(* Logix 5000 project; controller LeakTestAuto vendor 1 type 14 code 226 rev 37.11; software revision 37.01; part 14 of 15 *)
(* tags used below, declared in another part *)
   AOI_CapActuators_Seq : AOI_Sequencer_x64;
   AOI_CapCTS_Seq : AOI_Sequencer_x64;
   AOI_CapFail_Seq : AOI_Sequencer_x64;
   AOI_CapRobot_Seq : AOI_Sequencer_x64;
   AOI_CTS1 : AOI_CTS_INSTRUMENT;
   AOI_CTS2 : AOI_CTS_INSTRUMENT;
   AOI_RobotPos : AOI_RobotPositions;
   AOI_SeqSteps : AOI_StandardSeqSteps;
   AOI_SRX100 : AOI_KeyenceBarcode;
   BarcodeScanner : udt_OutputStructure;
   CapActuators_BarcodeBad : COUNTER;
   CapActuators_BarcodeGood : COUNTER;
   CapActuators_CTS1Bad : COUNTER;
   CapActuators_CTS1Good : COUNTER;
   CapActuators_CTS2Bad : COUNTER;
   CapActuators_CTS2Good : COUNTER;
   CapActuators_Nest1HasPart : BOOL;
   CapActuators_Nest2HasPart : BOOL;
   CapActuators_Seq : udt_SequenceStructure_X64;
   CapCTS_CTS1Bad : COUNTER;
   CapCTS_CTS1Good : COUNTER;
   CapCTS_CTS2Bad : COUNTER;
   CapCTS_CTS2Good : COUNTER;
   CapCTS_Nest1HasPart : BOOL;
   CapCTS_Nest2HasPart : BOOL;
   CapCTS_Seq : udt_SequenceStructure_X64;
   CapFail_Seq : udt_SequenceStructure_X64;
   CapRobot_IsNest : BOOL;
   CapRobot_Seq : udt_SequenceStructure_X64;
   CapRobot_StartPos : DINT;
   CapRobot_TargetPos : DINT;
   CapShuffle_Seq : udt_SequenceStructure_X64;
   Conveyor : udt_OutputStructure;
   Conveyor_Seq : udt_SequenceStructure_X64;
   LeakTester1 : udt_OutputStructure;
   LeakTester2 : udt_OutputStructure;
   Nest1Cylinder : udt_OutputStructure;
   Nest2Cylinder : udt_OutputStructure;
   OP220 : udt_Mode;
   Robot : udt_OutputStructure;
   RobotGripper : udt_OutputStructure;
   RobotInputs : udt_EpsonInputs;
   TempConsumedFromPLC : BOOL;
   TON_CapActuatorsDelay : TIMER;
   TON_CapActuatorsDelay2 : TIMER;
   TON_CapCTSDelay : TIMER;
   TON_CapCTSDelay2 : TIMER;
   TON_FailChute : TIMER[10];
   I_OP220_N3_CONVEYOR_LOAD : ALIAS FOR Local:3:I.Pt12.Data;
   I_OP220_N3_DUT_PRE_NEST_0 : ALIAS FOR Local:3:I.Pt00.Data;
   I_OP220_N3_DUT_PRE_NEST_1 : ALIAS FOR Local:3:I.Pt01.Data;
   I_OP220_N3_DUT_PRE_NEST_2 : ALIAS FOR Local:3:I.Pt02.Data;
   I_OP220_N3_NEST1_EXTEND : ALIAS FOR Local:3:I.Pt04.Data;
   I_OP220_N3_NEST1_HOME : ALIAS FOR Local:3:I.Pt03.Data;
   I_OP220_N3_NEST2_EXTEND : ALIAS FOR Local:3:I.Pt06.Data;
   I_OP220_N3_NEST2_HOME : ALIAS FOR Local:3:I.Pt05.Data;
   I_OP220_N3_REJECT_CHUTE_PART : ALIAS FOR Local:3:I.Pt10.Data;
   PLC : AOI_PLC;
(* MainProgram, continued *)

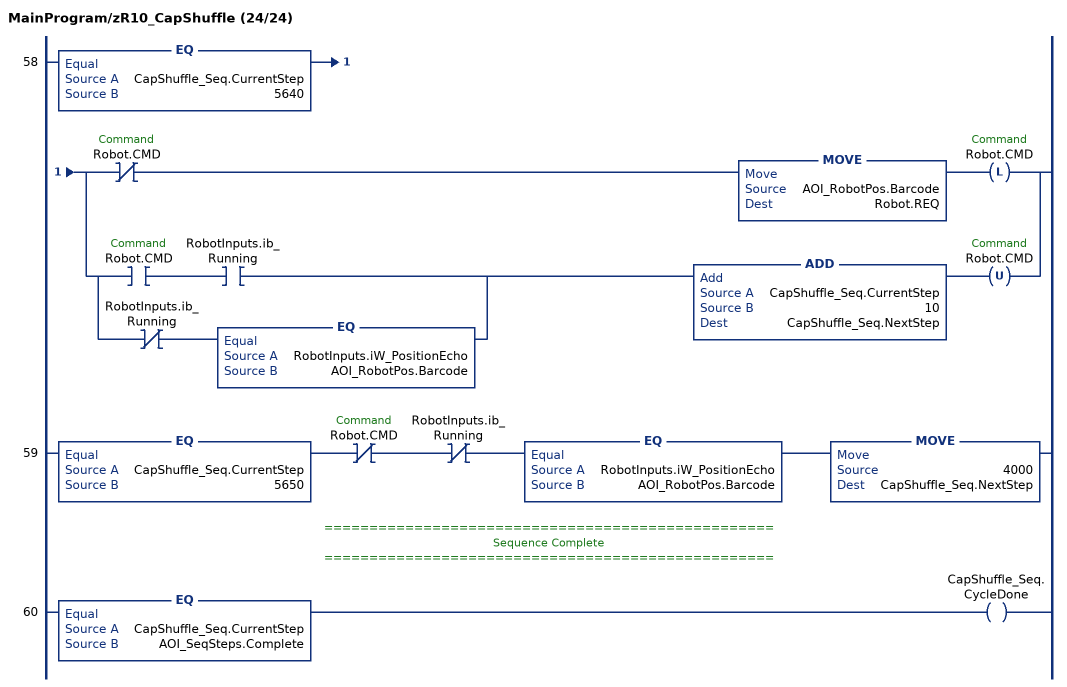
   [picture p173: MainProgram/zR10_CapShuffle rungs 58-60]
   58: EQ(CapShuffle_Seq.CurrentStep,5640)[XIO(Robot.CMD) MOVE(AOI_RobotPos.Barcode,Robot.REQ) OTL(Robot.CMD) ,[XIC(Robot.CMD) XIC(RobotInputs.ib_Running) ,XIO(RobotInputs.ib_Running) EQ(RobotInputs.iW_PositionEcho,AOI_RobotPos.Barcode) ] ADD(CapShuffle_Seq.CurrentStep,10,CapShuffle_Seq.NextStep) OTU(Robot.CMD) ];
   59: EQ(CapShuffle_Seq.CurrentStep,5650)XIO(Robot.CMD)XIO(RobotInputs.ib_Running)EQ(RobotInputs.iW_PositionEcho,AOI_RobotPos.Barcode)MOVE(4000,CapShuffle_Seq.NextStep);
   // ==================================================
   // Sequence Complete
   // ==================================================
   60: EQ(CapShuffle_Seq.CurrentStep,AOI_SeqSteps.Complete)OTE(CapShuffle_Seq.CycleDone);
END_ROUTINE

ROUTINE zR20_CapActuators   (* ladder *)
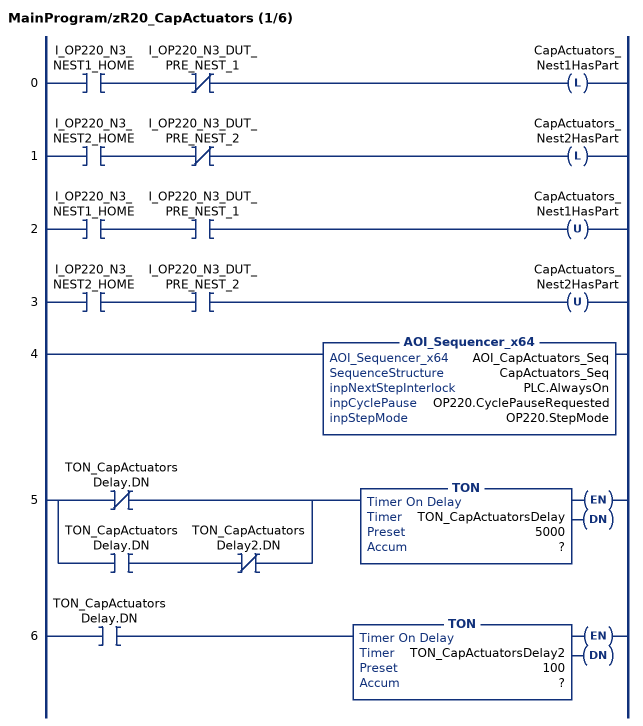
   0: XIC(I_OP220_N3_NEST1_HOME)XIO(I_OP220_N3_DUT_PRE_NEST_1)OTL(CapActuators_Nest1HasPart);
   1: XIC(I_OP220_N3_NEST2_HOME)XIO(I_OP220_N3_DUT_PRE_NEST_2)OTL(CapActuators_Nest2HasPart);
   2: XIC(I_OP220_N3_NEST1_HOME)XIC(I_OP220_N3_DUT_PRE_NEST_1)OTU(CapActuators_Nest1HasPart);
   3: XIC(I_OP220_N3_NEST2_HOME)XIC(I_OP220_N3_DUT_PRE_NEST_2)OTU(CapActuators_Nest2HasPart);
   4: AOI_Sequencer_x64(AOI_CapActuators_Seq,CapActuators_Seq,PLC.AlwaysOn,OP220.CyclePauseRequested,OP220.StepMode);
   5: [XIO(TON_CapActuatorsDelay.DN) ,XIC(TON_CapActuatorsDelay.DN) XIO(TON_CapActuatorsDelay2.DN) ]TON(TON_CapActuatorsDelay,?,?);
   6: XIC(TON_CapActuatorsDelay.DN)TON(TON_CapActuatorsDelay2,?,?);
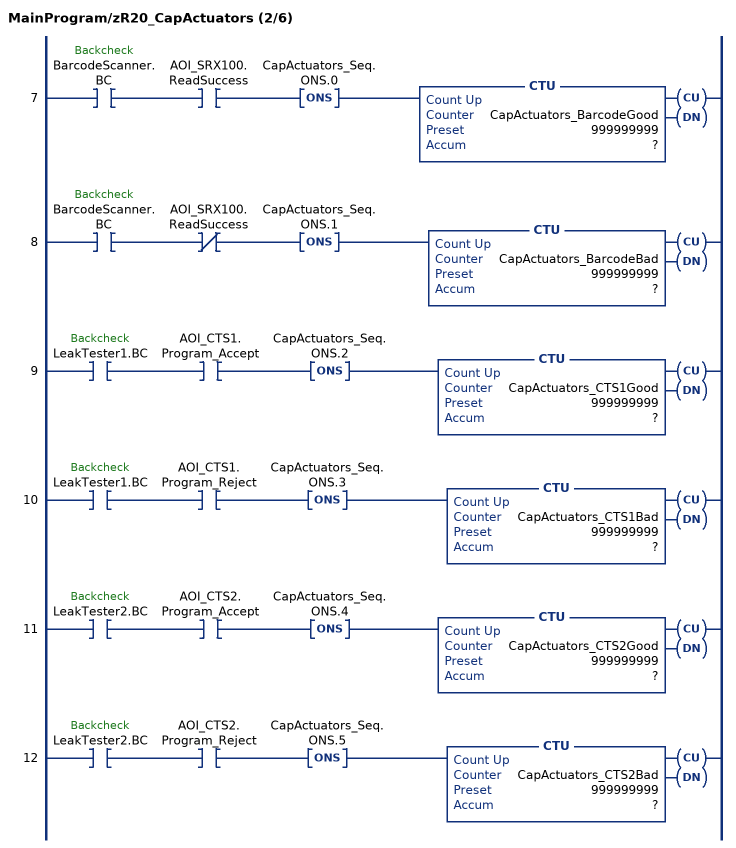
   7: XIC(BarcodeScanner.BC)XIC(AOI_SRX100.ReadSuccess)ONS(CapActuators_Seq.ONS.0)CTU(CapActuators_BarcodeGood,?,?);
   8: XIC(BarcodeScanner.BC)XIO(AOI_SRX100.ReadSuccess)ONS(CapActuators_Seq.ONS.1)CTU(CapActuators_BarcodeBad,?,?);
   9: XIC(LeakTester1.BC)XIC(AOI_CTS1.Program_Accept)ONS(CapActuators_Seq.ONS.2)CTU(CapActuators_CTS1Good,?,?);
   10: XIC(LeakTester1.BC)XIC(AOI_CTS1.Program_Reject)ONS(CapActuators_Seq.ONS.3)CTU(CapActuators_CTS1Bad,?,?);
   11: XIC(LeakTester2.BC)XIC(AOI_CTS2.Program_Accept)ONS(CapActuators_Seq.ONS.4)CTU(CapActuators_CTS2Good,?,?);
   12: XIC(LeakTester2.BC)XIC(AOI_CTS2.Program_Reject)ONS(CapActuators_Seq.ONS.5)CTU(CapActuators_CTS2Bad,?,?);
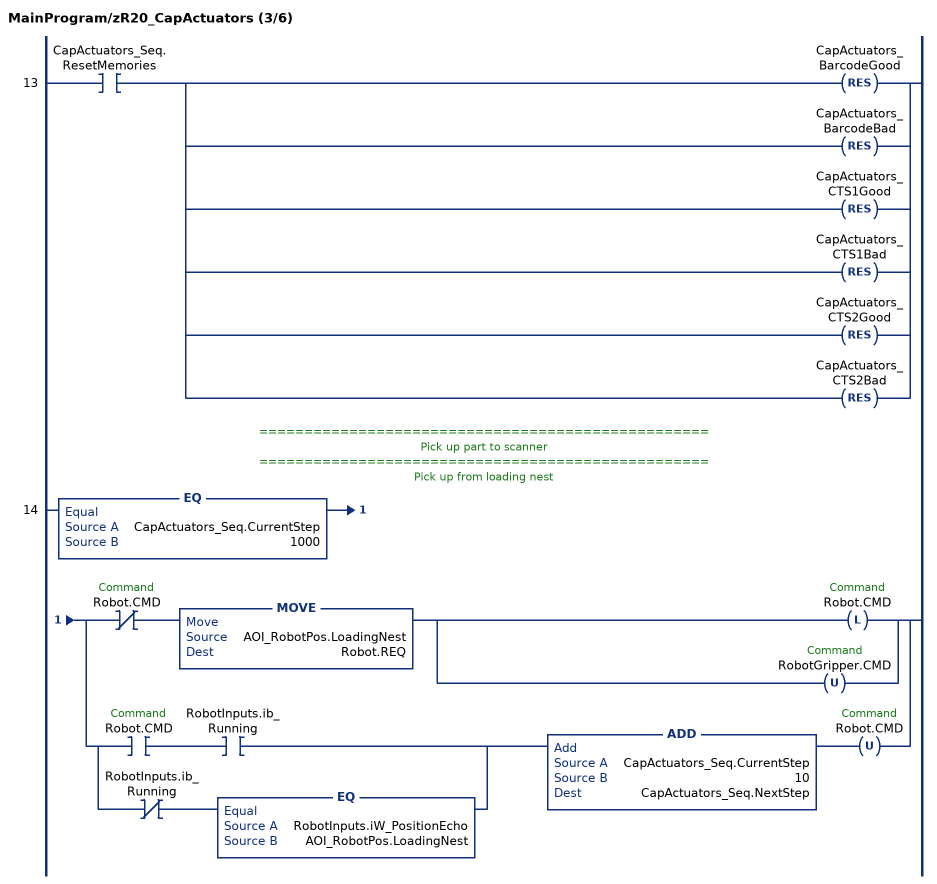
   13: XIC(CapActuators_Seq.ResetMemories)[RES(CapActuators_BarcodeGood) ,RES(CapActuators_BarcodeBad) ,RES(CapActuators_CTS1Good) ,RES(CapActuators_CTS1Bad) ,RES(CapActuators_CTS2Good) ,RES(CapActuators_CTS2Bad) ];
   // ==================================================
   // Pick up part to scanner
   // ==================================================
   // Pick up from loading nest
   14: EQ(CapActuators_Seq.CurrentStep,1000)[XIO(Robot.CMD) MOVE(AOI_RobotPos.LoadingNest,Robot.REQ) [OTL(Robot.CMD) ,OTU(RobotGripper.CMD) ] ,[XIC(Robot.CMD) XIC(RobotInputs.ib_Running) ,XIO(RobotInputs.ib_Running) EQ(RobotInputs.iW_PositionEcho,AOI_RobotPos.LoadingNest) ] ADD(CapActuators_Seq.CurrentStep,10,CapActuators_Seq.NextStep) OTU(Robot.CMD) ];
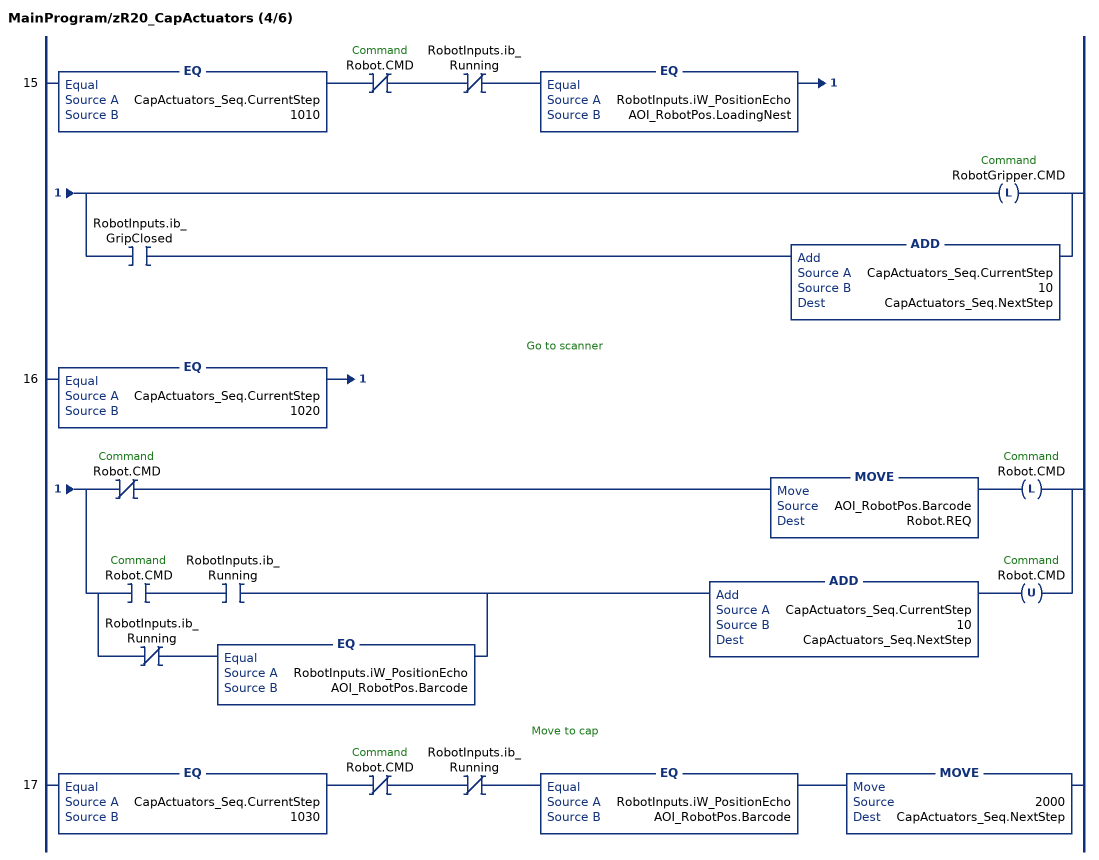
   15: EQ(CapActuators_Seq.CurrentStep,1010)XIO(Robot.CMD)XIO(RobotInputs.ib_Running)EQ(RobotInputs.iW_PositionEcho,AOI_RobotPos.LoadingNest)[OTL(RobotGripper.CMD) ,XIC(RobotInputs.ib_GripClosed) ADD(CapActuators_Seq.CurrentStep,10,CapActuators_Seq.NextStep) ];
   // Go to scanner
   16: EQ(CapActuators_Seq.CurrentStep,1020)[XIO(Robot.CMD) MOVE(AOI_RobotPos.Barcode,Robot.REQ) OTL(Robot.CMD) ,[XIC(Robot.CMD) XIC(RobotInputs.ib_Running) ,XIO(RobotInputs.ib_Running) EQ(RobotInputs.iW_PositionEcho,AOI_RobotPos.Barcode) ] ADD(CapActuators_Seq.CurrentStep,10,CapActuators_Seq.NextStep) OTU(Robot.CMD) ];
   // Move to cap
   17: EQ(CapActuators_Seq.CurrentStep,1030)XIO(Robot.CMD)XIO(RobotInputs.ib_Running)EQ(RobotInputs.iW_PositionEcho,AOI_RobotPos.Barcode)MOVE(2000,CapActuators_Seq.NextStep);
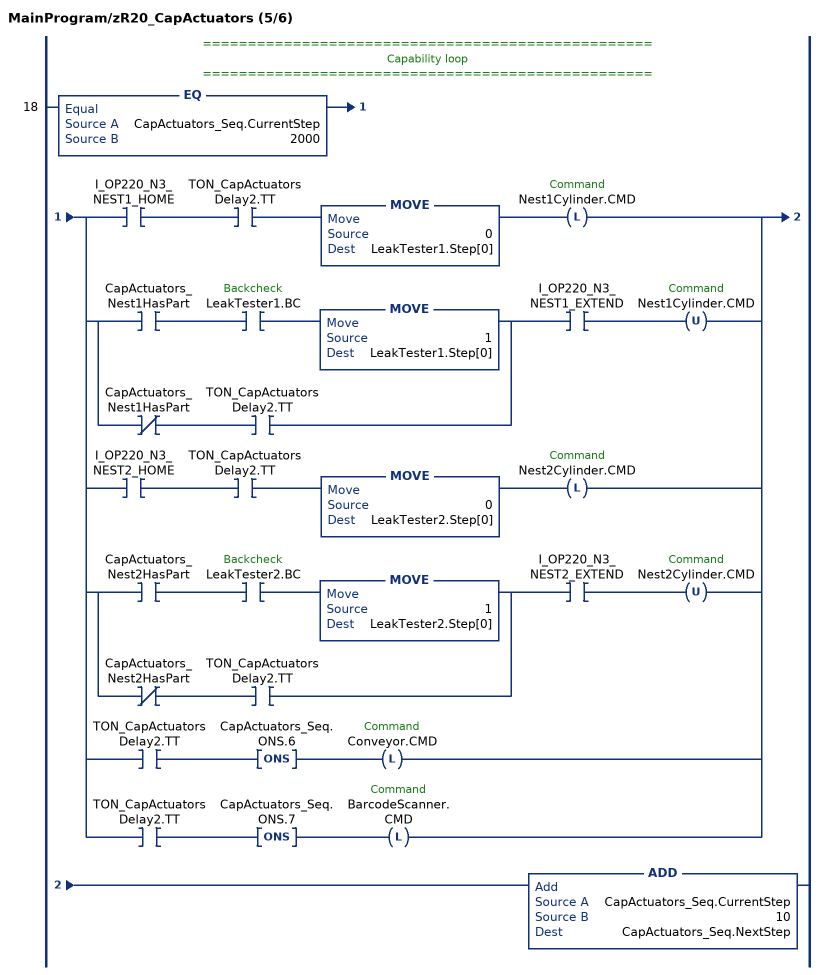
   // ==================================================
   // Capability loop
   // ==================================================
   18: EQ(CapActuators_Seq.CurrentStep,2000)[XIC(I_OP220_N3_NEST1_HOME) XIC(TON_CapActuatorsDelay2.TT) MOVE(0,LeakTester1.Step[0]) OTL(Nest1Cylinder.CMD) ,[XIC(CapActuators_Nest1HasPart) XIC(LeakTester1.BC) MOVE(1,LeakTester1.Step[0]) ,XIO(CapActuators_Nest1HasPart) XIC(TON_CapActuatorsDelay2.TT) ] XIC(I_OP220_N3_NEST1_EXTEND) OTU(Nest1Cylinder.CMD) ,XIC(I_OP220_N3_NEST2_HOME) XIC(TON_CapActuatorsDelay2.TT) MOVE(0,LeakTester2.Step[0]) OTL(Nest2Cylinder.CMD) ,[XIC(CapActuators_Nest2HasPart) XIC(LeakTester2.BC) MOVE(1,LeakTester2.Step[0]) ,XIO(CapActuators_Nest2HasPart) XIC(TON_CapActuatorsDelay2.TT) ] XIC(I_OP220_N3_NEST2_EXTEND) OTU(Nest2Cylinder.CMD) ,XIC(TON_CapActuatorsDelay2.TT) ONS(CapActuators_Seq.ONS.6) OTL(Conveyor.CMD) ,XIC(TON_CapActuatorsDelay2.TT) ONS(CapActuators_Seq.ONS.7) OTL(BarcodeScanner.CMD) ]ADD(CapActuators_Seq.CurrentStep,10,CapActuators_Seq.NextStep);
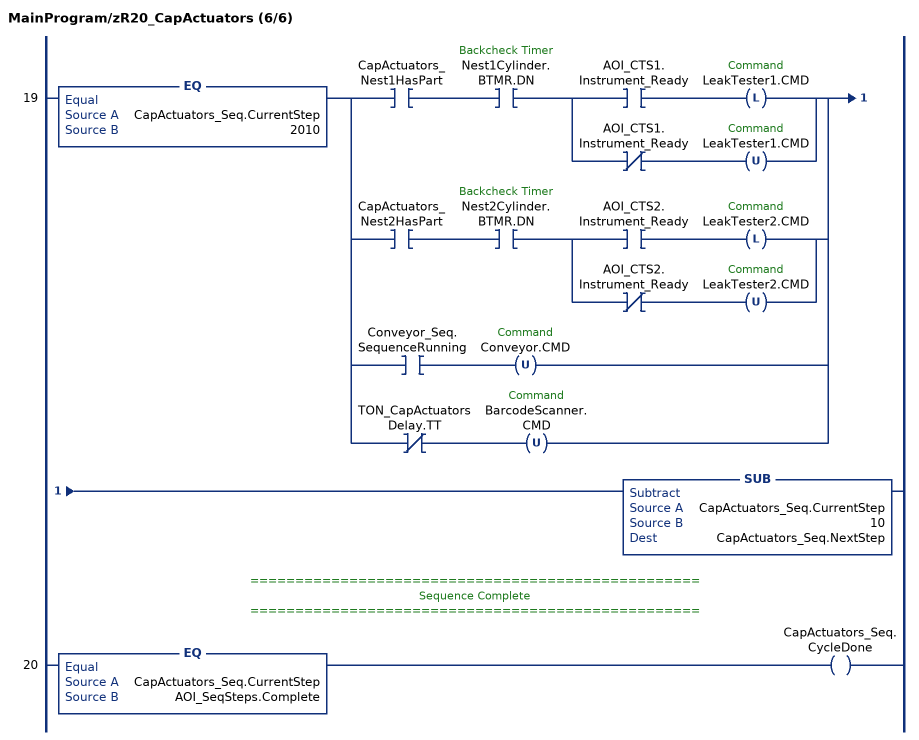
   19: EQ(CapActuators_Seq.CurrentStep,2010)[XIC(CapActuators_Nest1HasPart) XIC(Nest1Cylinder.BTMR.DN) [XIC(AOI_CTS1.Instrument_Ready) OTL(LeakTester1.CMD) ,XIO(AOI_CTS1.Instrument_Ready) OTU(LeakTester1.CMD) ] ,XIC(CapActuators_Nest2HasPart) XIC(Nest2Cylinder.BTMR.DN) [XIC(AOI_CTS2.Instrument_Ready) OTL(LeakTester2.CMD) ,XIO(AOI_CTS2.Instrument_Ready) OTU(LeakTester2.CMD) ] ,XIC(Conveyor_Seq.SequenceRunning) OTU(Conveyor.CMD) ,XIO(TON_CapActuatorsDelay.TT) OTU(BarcodeScanner.CMD) ]SUB(CapActuators_Seq.CurrentStep,10,CapActuators_Seq.NextStep);
   // ==================================================
   // Sequence Complete
   // ==================================================
   20: EQ(CapActuators_Seq.CurrentStep,AOI_SeqSteps.Complete)OTE(CapActuators_Seq.CycleDone);
END_ROUTINE

ROUTINE zR30_CapRobot   (* ladder *)
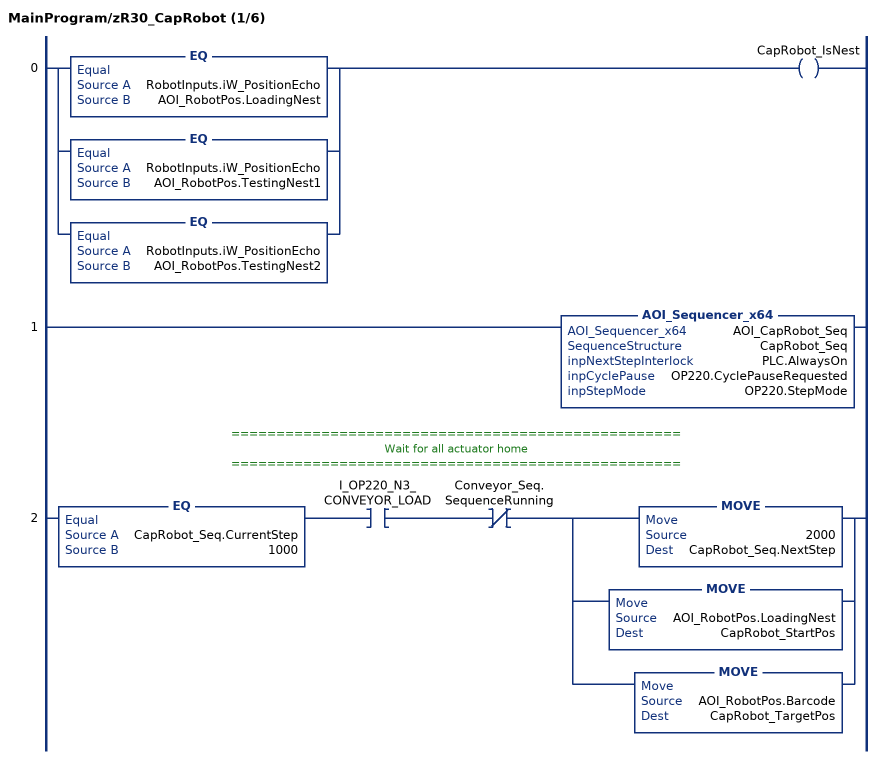
   0: [EQ(RobotInputs.iW_PositionEcho,AOI_RobotPos.LoadingNest) ,EQ(RobotInputs.iW_PositionEcho,AOI_RobotPos.TestingNest1) ,EQ(RobotInputs.iW_PositionEcho,AOI_RobotPos.TestingNest2) ]OTE(CapRobot_IsNest);
   1: AOI_Sequencer_x64(AOI_CapRobot_Seq,CapRobot_Seq,PLC.AlwaysOn,OP220.CyclePauseRequested,OP220.StepMode);
   // ==================================================
   // Wait for all actuator home
   // ==================================================
   2: EQ(CapRobot_Seq.CurrentStep,1000)XIC(I_OP220_N3_CONVEYOR_LOAD)XIO(Conveyor_Seq.SequenceRunning)[MOVE(2000,CapRobot_Seq.NextStep) ,MOVE(AOI_RobotPos.LoadingNest,CapRobot_StartPos) ,MOVE(AOI_RobotPos.Barcode,CapRobot_TargetPos) ];
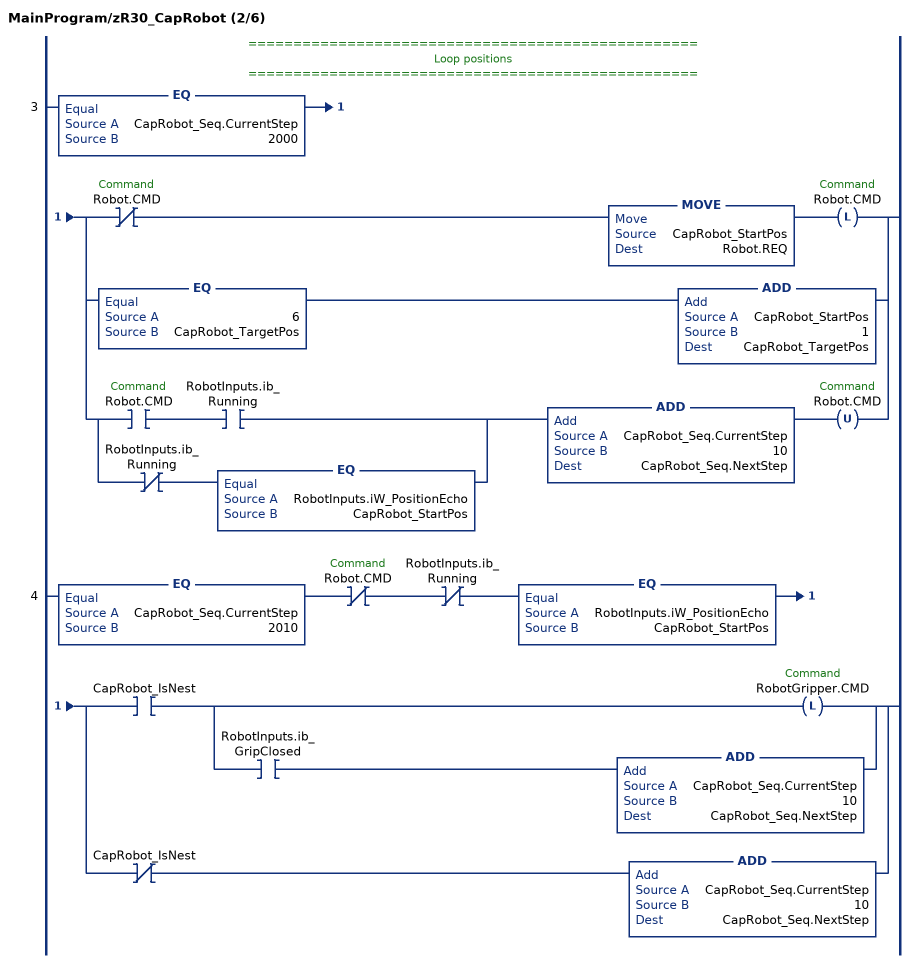
   // ==================================================
   // Loop positions
   // ==================================================
   3: EQ(CapRobot_Seq.CurrentStep,2000)[XIO(Robot.CMD) MOVE(CapRobot_StartPos,Robot.REQ) OTL(Robot.CMD) ,EQ(6,CapRobot_TargetPos) ADD(CapRobot_StartPos,1,CapRobot_TargetPos) ,[XIC(Robot.CMD) XIC(RobotInputs.ib_Running) ,XIO(RobotInputs.ib_Running) EQ(RobotInputs.iW_PositionEcho,CapRobot_StartPos) ] ADD(CapRobot_Seq.CurrentStep,10,CapRobot_Seq.NextStep) OTU(Robot.CMD) ];
   4: EQ(CapRobot_Seq.CurrentStep,2010)XIO(Robot.CMD)XIO(RobotInputs.ib_Running)EQ(RobotInputs.iW_PositionEcho,CapRobot_StartPos)[XIC(CapRobot_IsNest) [OTL(RobotGripper.CMD) ,XIC(RobotInputs.ib_GripClosed) ADD(CapRobot_Seq.CurrentStep,10,CapRobot_Seq.NextStep) ] ,XIO(CapRobot_IsNest) ADD(CapRobot_Seq.CurrentStep,10,CapRobot_Seq.NextStep) ];
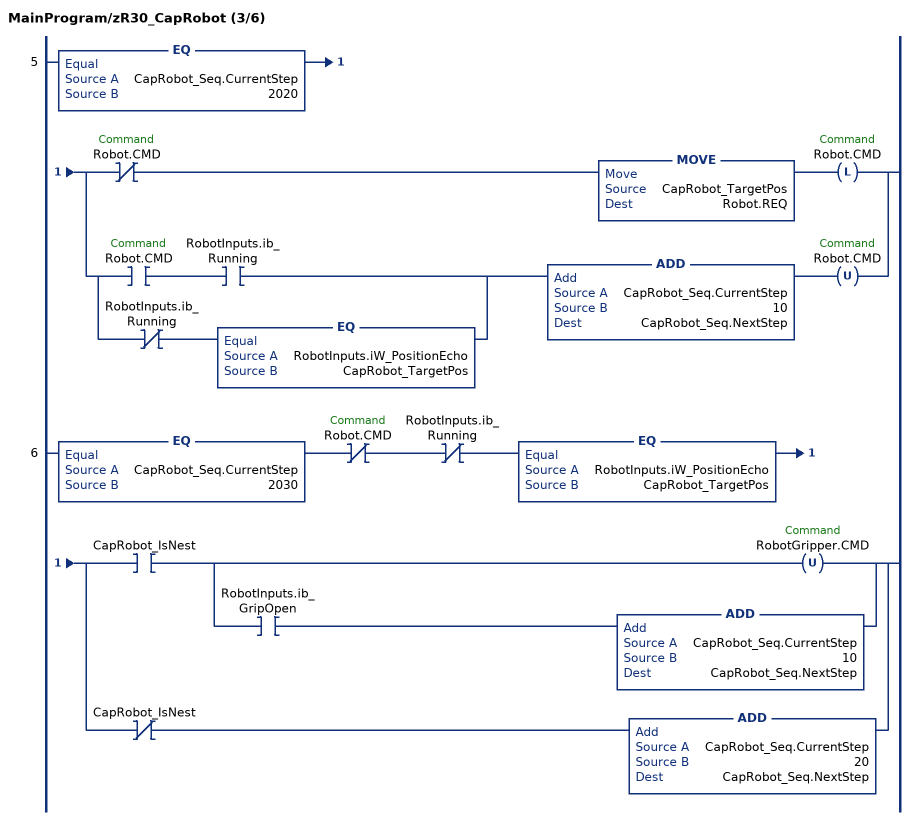
   5: EQ(CapRobot_Seq.CurrentStep,2020)[XIO(Robot.CMD) MOVE(CapRobot_TargetPos,Robot.REQ) OTL(Robot.CMD) ,[XIC(Robot.CMD) XIC(RobotInputs.ib_Running) ,XIO(RobotInputs.ib_Running) EQ(RobotInputs.iW_PositionEcho,CapRobot_TargetPos) ] ADD(CapRobot_Seq.CurrentStep,10,CapRobot_Seq.NextStep) OTU(Robot.CMD) ];
   6: EQ(CapRobot_Seq.CurrentStep,2030)XIO(Robot.CMD)XIO(RobotInputs.ib_Running)EQ(RobotInputs.iW_PositionEcho,CapRobot_TargetPos)[XIC(CapRobot_IsNest) [OTU(RobotGripper.CMD) ,XIC(RobotInputs.ib_GripOpen) ADD(CapRobot_Seq.CurrentStep,10,CapRobot_Seq.NextStep) ] ,XIO(CapRobot_IsNest) ADD(CapRobot_Seq.CurrentStep,20,CapRobot_Seq.NextStep) ];
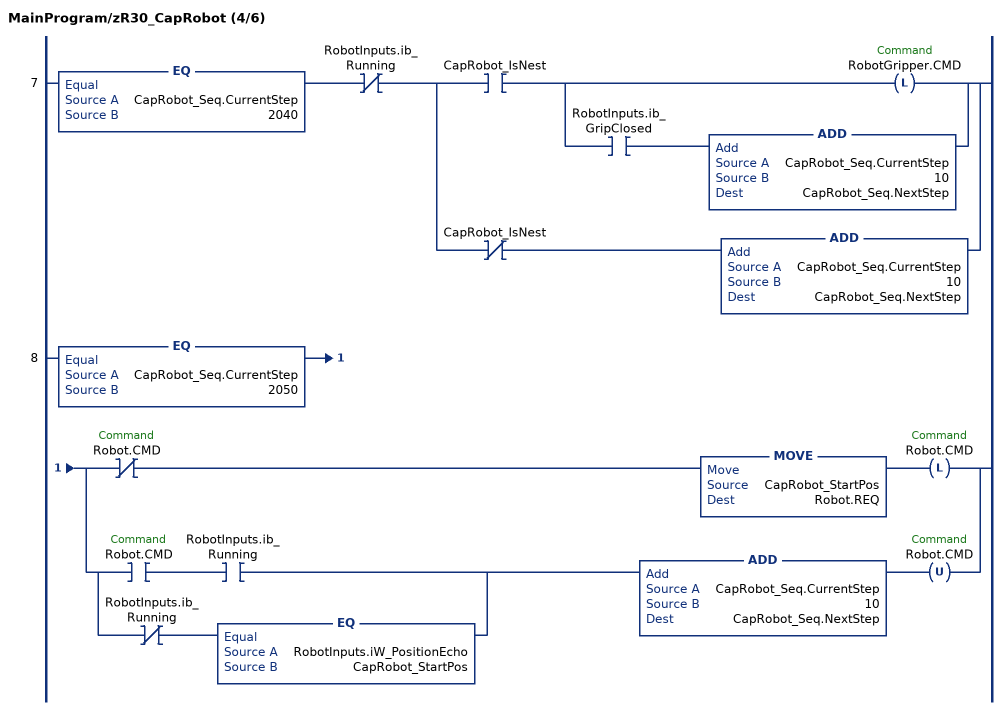
   7: EQ(CapRobot_Seq.CurrentStep,2040)XIO(RobotInputs.ib_Running)[XIC(CapRobot_IsNest) [OTL(RobotGripper.CMD) ,XIC(RobotInputs.ib_GripClosed) ADD(CapRobot_Seq.CurrentStep,10,CapRobot_Seq.NextStep) ] ,XIO(CapRobot_IsNest) ADD(CapRobot_Seq.CurrentStep,10,CapRobot_Seq.NextStep) ];
   8: EQ(CapRobot_Seq.CurrentStep,2050)[XIO(Robot.CMD) MOVE(CapRobot_StartPos,Robot.REQ) OTL(Robot.CMD) ,[XIC(Robot.CMD) XIC(RobotInputs.ib_Running) ,XIO(RobotInputs.ib_Running) EQ(RobotInputs.iW_PositionEcho,CapRobot_StartPos) ] ADD(CapRobot_Seq.CurrentStep,10,CapRobot_Seq.NextStep) OTU(Robot.CMD) ];
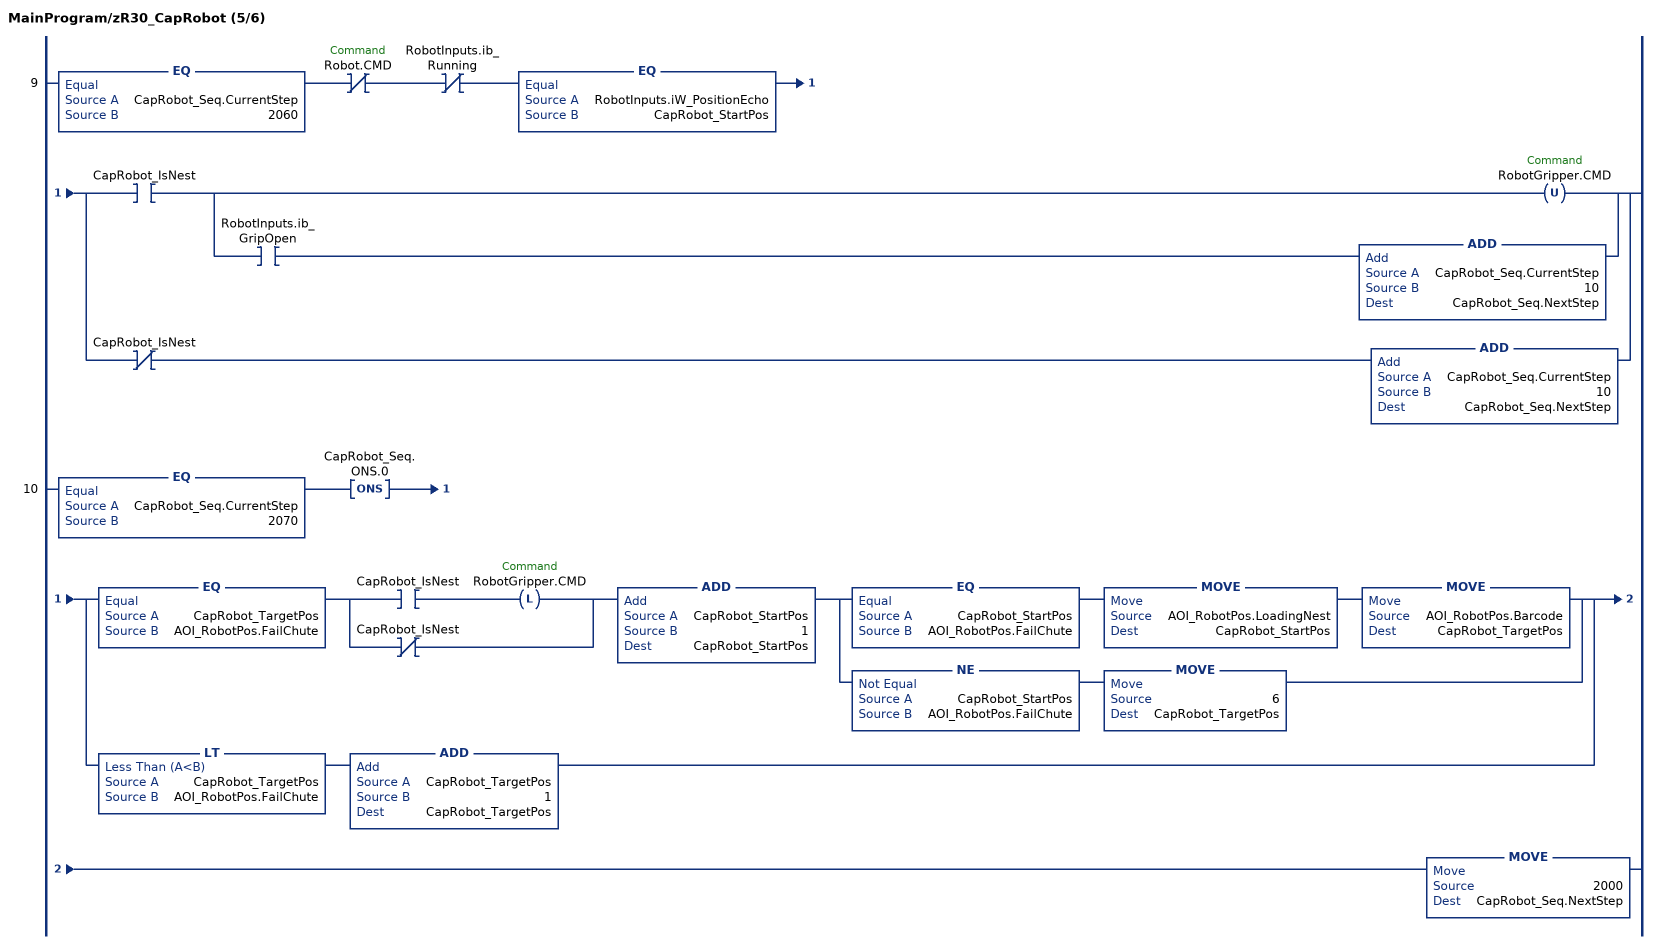
   9: EQ(CapRobot_Seq.CurrentStep,2060)XIO(Robot.CMD)XIO(RobotInputs.ib_Running)EQ(RobotInputs.iW_PositionEcho,CapRobot_StartPos)[XIC(CapRobot_IsNest) [OTU(RobotGripper.CMD) ,XIC(RobotInputs.ib_GripOpen) ADD(CapRobot_Seq.CurrentStep,10,CapRobot_Seq.NextStep) ] ,XIO(CapRobot_IsNest) ADD(CapRobot_Seq.CurrentStep,10,CapRobot_Seq.NextStep) ];
   10: EQ(CapRobot_Seq.CurrentStep,2070)ONS(CapRobot_Seq.ONS.0)[EQ(CapRobot_TargetPos,AOI_RobotPos.FailChute) [XIC(CapRobot_IsNest) OTL(RobotGripper.CMD) ,XIO(CapRobot_IsNest) ] ADD(CapRobot_StartPos,1,CapRobot_StartPos) [EQ(CapRobot_StartPos,AOI_RobotPos.FailChute) MOVE(AOI_RobotPos.LoadingNest,CapRobot_StartPos) MOVE(AOI_RobotPos.Barcode,CapRobot_TargetPos) ,NE(CapRobot_StartPos,AOI_RobotPos.FailChute) MOVE(6,CapRobot_TargetPos) ] ,LT(CapRobot_TargetPos,AOI_RobotPos.FailChute) ADD(CapRobot_TargetPos,1,CapRobot_TargetPos) ]MOVE(2000,CapRobot_Seq.NextStep);
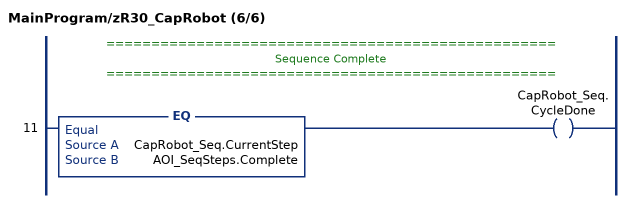
   // ==================================================
   // Sequence Complete
   // ==================================================
   11: EQ(CapRobot_Seq.CurrentStep,AOI_SeqSteps.Complete)OTE(CapRobot_Seq.CycleDone);
END_ROUTINE

ROUTINE zR40_CapCTS   (* ladder *)
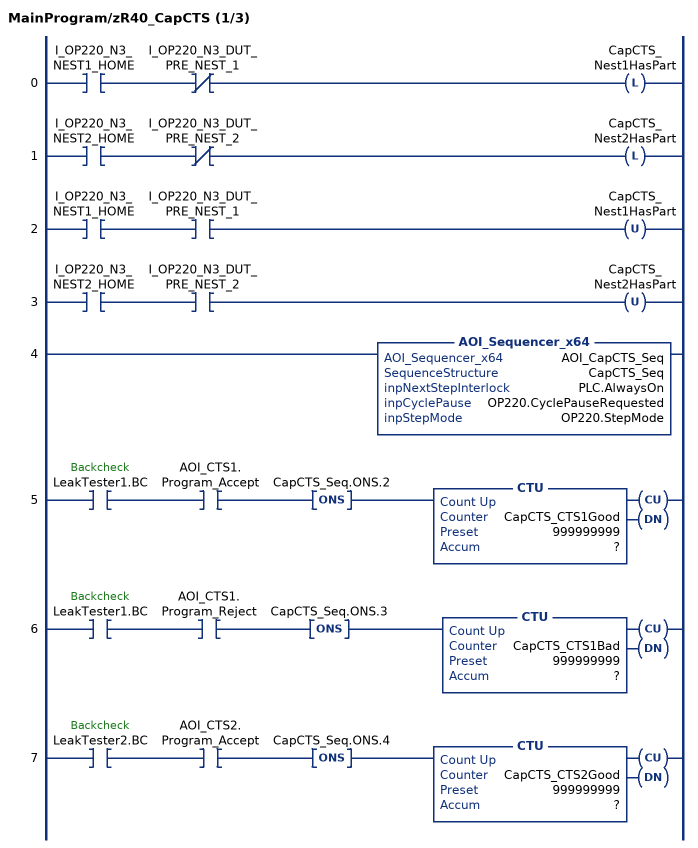
   0: XIC(I_OP220_N3_NEST1_HOME)XIO(I_OP220_N3_DUT_PRE_NEST_1)OTL(CapCTS_Nest1HasPart);
   1: XIC(I_OP220_N3_NEST2_HOME)XIO(I_OP220_N3_DUT_PRE_NEST_2)OTL(CapCTS_Nest2HasPart);
   2: XIC(I_OP220_N3_NEST1_HOME)XIC(I_OP220_N3_DUT_PRE_NEST_1)OTU(CapCTS_Nest1HasPart);
   3: XIC(I_OP220_N3_NEST2_HOME)XIC(I_OP220_N3_DUT_PRE_NEST_2)OTU(CapCTS_Nest2HasPart);
   4: AOI_Sequencer_x64(AOI_CapCTS_Seq,CapCTS_Seq,PLC.AlwaysOn,OP220.CyclePauseRequested,OP220.StepMode);
   5: XIC(LeakTester1.BC)XIC(AOI_CTS1.Program_Accept)ONS(CapCTS_Seq.ONS.2)CTU(CapCTS_CTS1Good,?,?);
   6: XIC(LeakTester1.BC)XIC(AOI_CTS1.Program_Reject)ONS(CapCTS_Seq.ONS.3)CTU(CapCTS_CTS1Bad,?,?);
   7: XIC(LeakTester2.BC)XIC(AOI_CTS2.Program_Accept)ONS(CapCTS_Seq.ONS.4)CTU(CapCTS_CTS2Good,?,?);
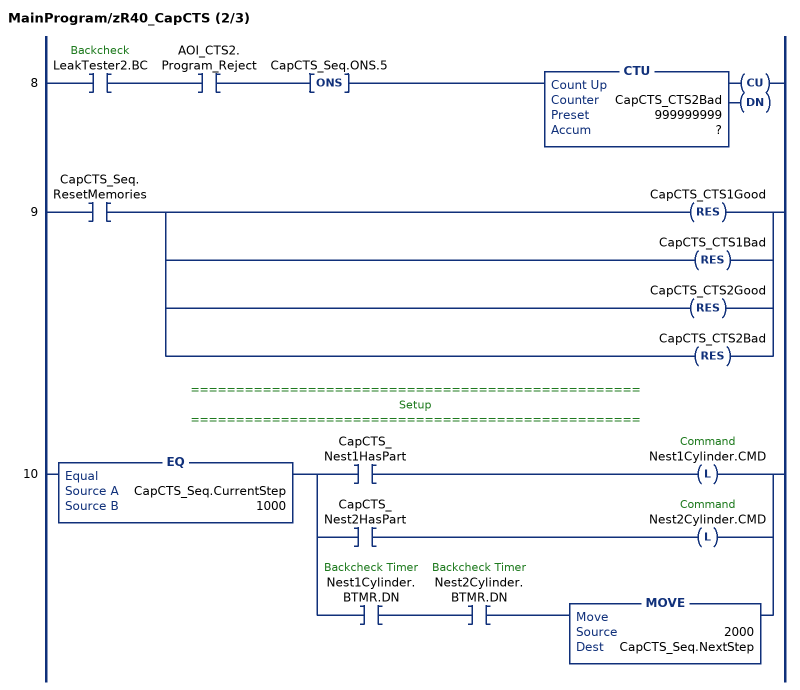
   8: XIC(LeakTester2.BC)XIC(AOI_CTS2.Program_Reject)ONS(CapCTS_Seq.ONS.5)CTU(CapCTS_CTS2Bad,?,?);
   9: XIC(CapCTS_Seq.ResetMemories)[RES(CapCTS_CTS1Good) ,RES(CapCTS_CTS1Bad) ,RES(CapCTS_CTS2Good) ,RES(CapCTS_CTS2Bad) ];
   // ==================================================
   // Setup
   // ==================================================
   10: EQ(CapCTS_Seq.CurrentStep,1000)[XIC(CapCTS_Nest1HasPart) OTL(Nest1Cylinder.CMD) ,XIC(CapCTS_Nest2HasPart) OTL(Nest2Cylinder.CMD) ,XIC(Nest1Cylinder.BTMR.DN) XIC(Nest2Cylinder.BTMR.DN) MOVE(2000,CapCTS_Seq.NextStep) ];
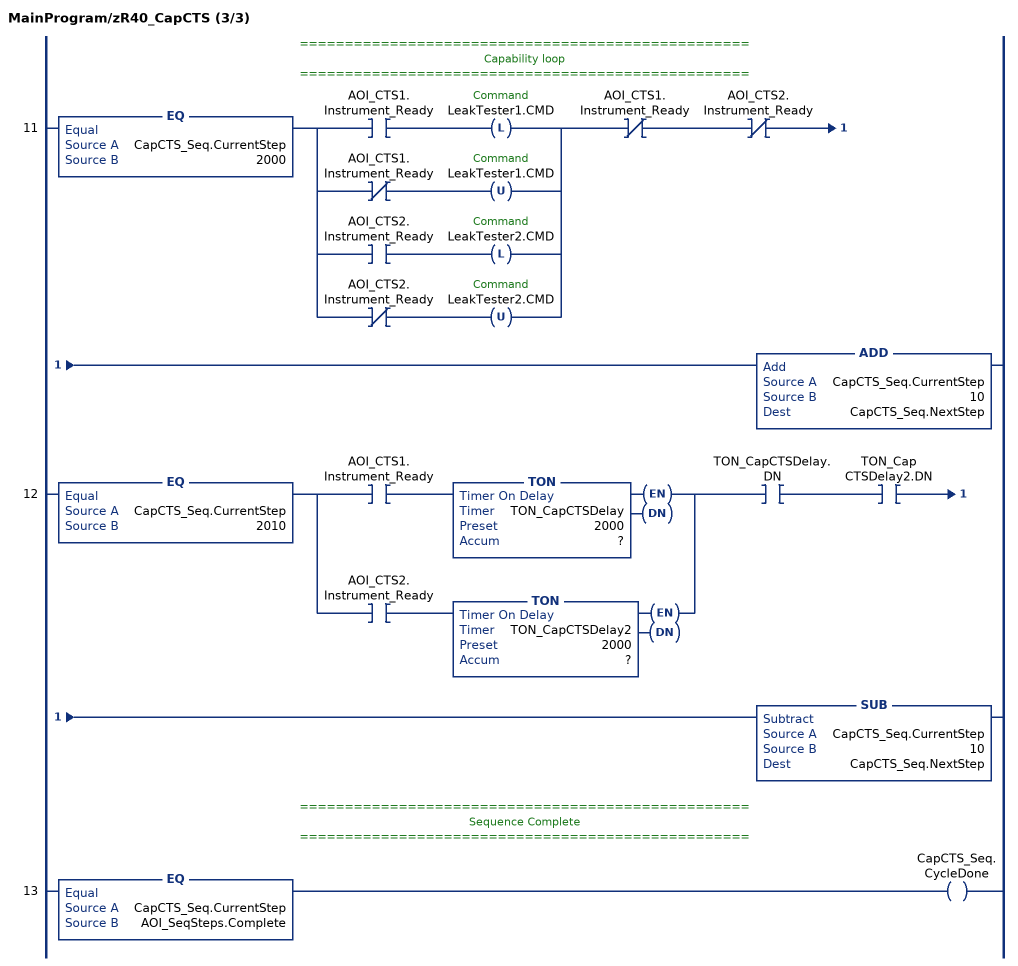
   // ==================================================
   // Capability loop
   // ==================================================
   11: EQ(CapCTS_Seq.CurrentStep,2000)[XIC(AOI_CTS1.Instrument_Ready) OTL(LeakTester1.CMD) ,XIO(AOI_CTS1.Instrument_Ready) OTU(LeakTester1.CMD) ,XIC(AOI_CTS2.Instrument_Ready) OTL(LeakTester2.CMD) ,XIO(AOI_CTS2.Instrument_Ready) OTU(LeakTester2.CMD) ]XIO(AOI_CTS1.Instrument_Ready)XIO(AOI_CTS2.Instrument_Ready)ADD(CapCTS_Seq.CurrentStep,10,CapCTS_Seq.NextStep);
   12: EQ(CapCTS_Seq.CurrentStep,2010)[XIC(AOI_CTS1.Instrument_Ready) TON(TON_CapCTSDelay,?,?) ,XIC(AOI_CTS2.Instrument_Ready) TON(TON_CapCTSDelay2,?,?) ]XIC(TON_CapCTSDelay.DN)XIC(TON_CapCTSDelay2.DN)SUB(CapCTS_Seq.CurrentStep,10,CapCTS_Seq.NextStep);
   // ==================================================
   // Sequence Complete
   // ==================================================
   13: EQ(CapCTS_Seq.CurrentStep,AOI_SeqSteps.Complete)OTE(CapCTS_Seq.CycleDone);
END_ROUTINE

ROUTINE zR50_CapFail   (* ladder *)
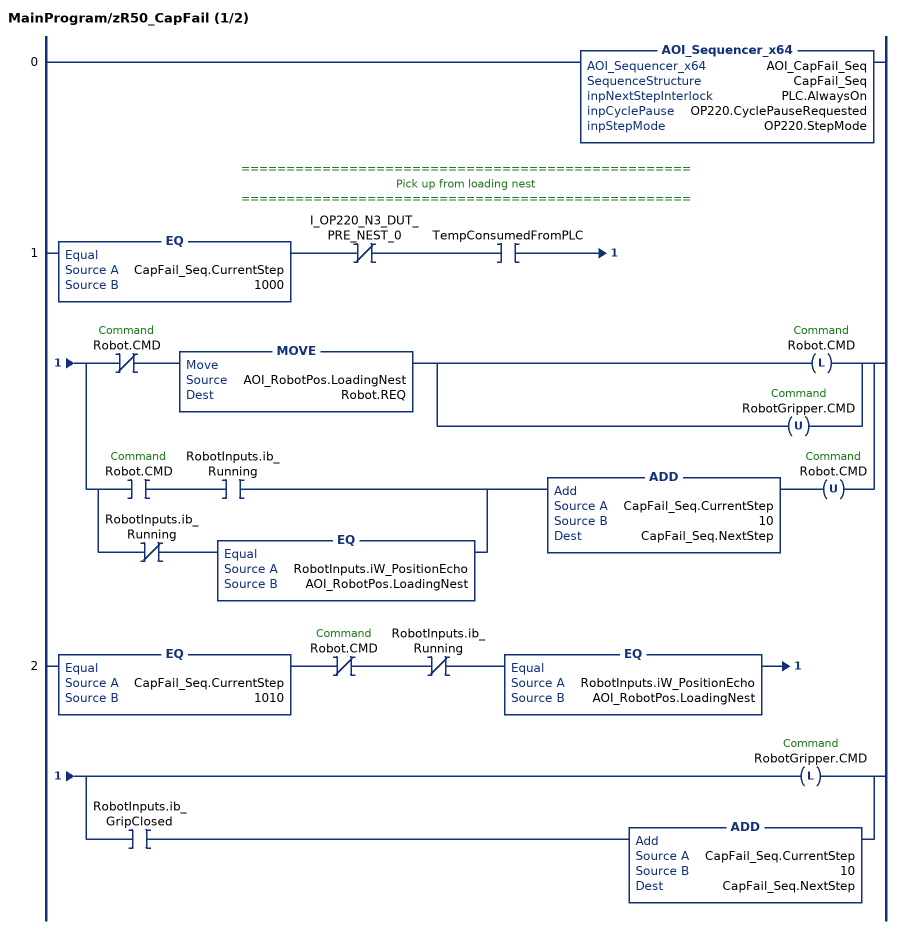
   0: AOI_Sequencer_x64(AOI_CapFail_Seq,CapFail_Seq,PLC.AlwaysOn,OP220.CyclePauseRequested,OP220.StepMode);
   // ==================================================
   // Pick up from loading nest
   // ==================================================
   1: EQ(CapFail_Seq.CurrentStep,1000)XIO(I_OP220_N3_DUT_PRE_NEST_0)XIC(TempConsumedFromPLC)[XIO(Robot.CMD) MOVE(AOI_RobotPos.LoadingNest,Robot.REQ) [OTL(Robot.CMD) ,OTU(RobotGripper.CMD) ] ,[XIC(Robot.CMD) XIC(RobotInputs.ib_Running) ,XIO(RobotInputs.ib_Running) EQ(RobotInputs.iW_PositionEcho,AOI_RobotPos.LoadingNest) ] ADD(CapFail_Seq.CurrentStep,10,CapFail_Seq.NextStep) OTU(Robot.CMD) ];
   2: EQ(CapFail_Seq.CurrentStep,1010)XIO(Robot.CMD)XIO(RobotInputs.ib_Running)EQ(RobotInputs.iW_PositionEcho,AOI_RobotPos.LoadingNest)[OTL(RobotGripper.CMD) ,XIC(RobotInputs.ib_GripClosed) ADD(CapFail_Seq.CurrentStep,10,CapFail_Seq.NextStep) ];
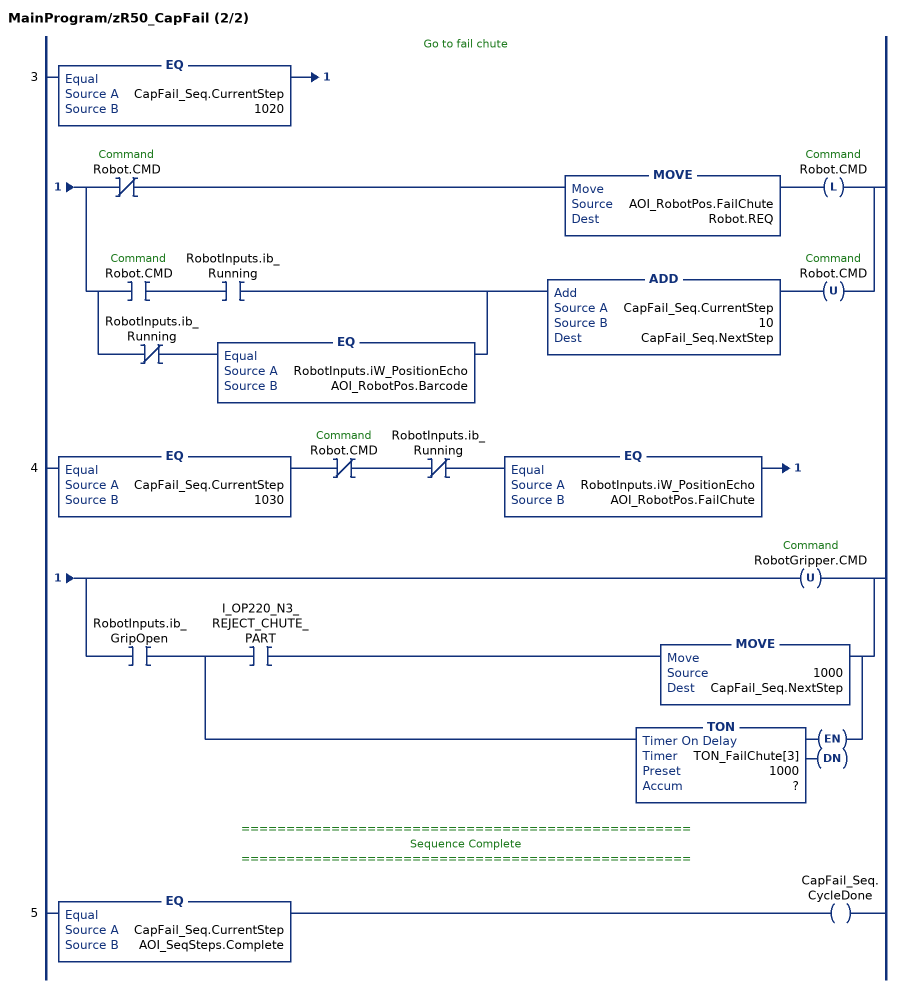
   // Go to fail chute
   3: EQ(CapFail_Seq.CurrentStep,1020)[XIO(Robot.CMD) MOVE(AOI_RobotPos.FailChute,Robot.REQ) OTL(Robot.CMD) ,[XIC(Robot.CMD) XIC(RobotInputs.ib_Running) ,XIO(RobotInputs.ib_Running) EQ(RobotInputs.iW_PositionEcho,AOI_RobotPos.Barcode) ] ADD(CapFail_Seq.CurrentStep,10,CapFail_Seq.NextStep) OTU(Robot.CMD) ];
   4: EQ(CapFail_Seq.CurrentStep,1030)XIO(Robot.CMD)XIO(RobotInputs.ib_Running)EQ(RobotInputs.iW_PositionEcho,AOI_RobotPos.FailChute)[OTU(RobotGripper.CMD) ,XIC(RobotInputs.ib_GripOpen) [XIC(I_OP220_N3_REJECT_CHUTE_PART) MOVE(1000,CapFail_Seq.NextStep) ,TON(TON_FailChute[3],?,?) ] ];
   // ==================================================
   // Sequence Complete
   // ==================================================
   5: EQ(CapFail_Seq.CurrentStep,AOI_SeqSteps.Complete)OTE(CapFail_Seq.CycleDone);
END_ROUTINE
